// TIA Portal V20 export
FUNCTION "04 T5 EXCENTRIC Transitions" : Void   // FC1418, LAD
TITLE = TRANSITIONS
{ S7_Optimized_Access := 'TRUE' }
// stored: AutoNumber false, SetENOAutomatically false
   VAR_TEMP
      Aux_real : Real;
   END_VAR
BEGIN

REGION Network 1: ============ TRANSITIONS ============
END_REGION

REGION Network 2: Transitions - Zone Status
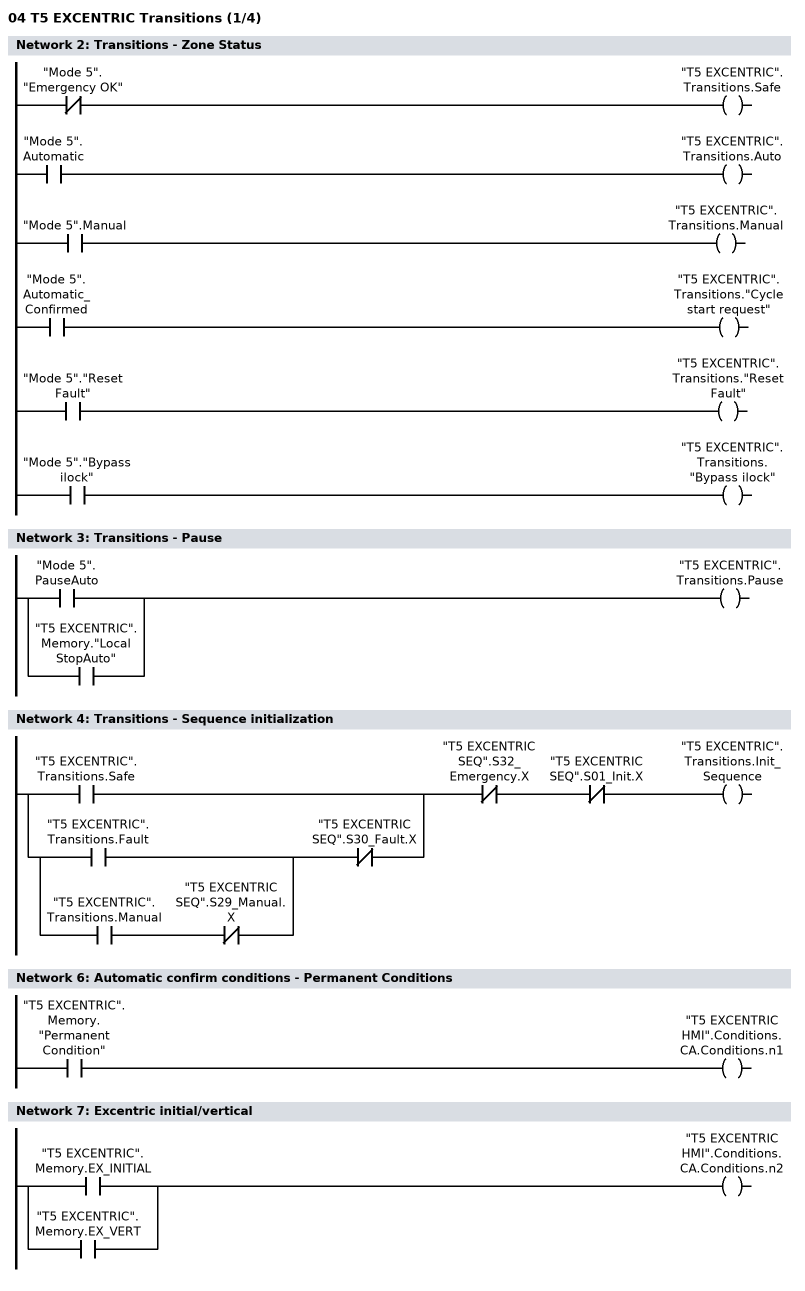
   RUNG wire#powerrail
      I_Contact( "Mode 5"."Emergency OK" )
      Coil( "T5 EXCENTRIC".Transitions.Safe )
   END_RUNG
   RUNG wire#powerrail
      Contact( "Mode 5".Automatic )
      Coil( "T5 EXCENTRIC".Transitions.Auto )
   END_RUNG
   RUNG wire#powerrail
      Contact( "Mode 5".Manual )
      Coil( "T5 EXCENTRIC".Transitions.Manual )
   END_RUNG
   RUNG wire#powerrail
      Contact( "Mode 5".Automatic_Confirmed )
      Coil( "T5 EXCENTRIC".Transitions."Cycle start request" )
   END_RUNG
   RUNG wire#powerrail
      Contact( "Mode 5"."Reset Fault" )
      Coil( "T5 EXCENTRIC".Transitions."Reset Fault" )
   END_RUNG
   RUNG wire#powerrail
      Contact( "Mode 5"."Bypass ilock" )
      Coil( "T5 EXCENTRIC".Transitions."Bypass ilock" )
   END_RUNG
   // the same network as SCL:
   "T5 EXCENTRIC".Transitions.Safe := NOT "Mode 5"."Emergency OK";
   "T5 EXCENTRIC".Transitions.Auto := "Mode 5".Automatic;
   "T5 EXCENTRIC".Transitions.Manual := "Mode 5".Manual;
   "T5 EXCENTRIC".Transitions."Cycle start request" := "Mode 5".Automatic_Confirmed;
   "T5 EXCENTRIC".Transitions."Reset Fault" := "Mode 5"."Reset Fault";
   "T5 EXCENTRIC".Transitions."Bypass ilock" := "Mode 5"."Bypass ilock";
END_REGION

REGION Network 3: Transitions - Pause
   RUNG wire#powerrail
      Contact( "Mode 5".PauseAuto )
      wire#w1
      Coil( "T5 EXCENTRIC".Transitions.Pause )
   END_RUNG
   RUNG wire#powerrail
      Contact( "T5 EXCENTRIC".Memory."Local StopAuto" )
   END_RUNG wire#w1
   // the same network as SCL:
   "T5 EXCENTRIC".Transitions.Pause := "Mode 5".PauseAuto OR "T5 EXCENTRIC".Memory."Local StopAuto";
END_REGION

REGION Network 4: Transitions - Sequence initialization
   RUNG wire#powerrail
      Contact( "T5 EXCENTRIC".Transitions.Safe )
      wire#w1
      I_Contact( "T5 EXCENTRIC SEQ".S32_Emergency.X )
      I_Contact( "T5 EXCENTRIC SEQ".S01_Init.X )
      Coil( "T5 EXCENTRIC".Transitions.Init_Sequence )
   END_RUNG
   RUNG wire#powerrail
      Contact( "T5 EXCENTRIC".Transitions.Fault )
      wire#w2
      I_Contact( "T5 EXCENTRIC SEQ".S30_Fault.X )
   END_RUNG wire#w1
   RUNG wire#powerrail
      Contact( "T5 EXCENTRIC".Transitions.Manual )
      I_Contact( "T5 EXCENTRIC SEQ".S29_Manual.X )
   END_RUNG wire#w2
   // the same network as SCL:
   "T5 EXCENTRIC".Transitions.Init_Sequence := ("T5 EXCENTRIC".Transitions.Safe OR (("T5 EXCENTRIC".Transitions.Fault OR ("T5 EXCENTRIC".Transitions.Manual AND NOT "T5 EXCENTRIC SEQ".S29_Manual.X)) AND NOT "T5 EXCENTRIC SEQ".S30_Fault.X)) AND NOT "T5 EXCENTRIC SEQ".S32_Emergency.X AND NOT "T5 EXCENTRIC SEQ".S01_Init.X;
END_REGION

REGION Network 5: ============ AUTOMATIC CONFIRM CONDITIONS - 1ST PIECE ============
END_REGION

REGION Network 6: Automatic confirm conditions - Permanent Conditions
   RUNG wire#powerrail
      Contact( "T5 EXCENTRIC".Memory."Permanent Condition" )
      Coil( "T5 EXCENTRIC HMI".Conditions.CA.Conditions.n1 )
   END_RUNG
   // the same network as SCL:
   "T5 EXCENTRIC HMI".Conditions.CA.Conditions.n1 := "T5 EXCENTRIC".Memory."Permanent Condition";
END_REGION

REGION Network 7: Excentric initial/vertical
   RUNG wire#powerrail
      Contact( "T5 EXCENTRIC".Memory.EX_INITIAL )
      wire#w1
      Coil( "T5 EXCENTRIC HMI".Conditions.CA.Conditions.n2 )
   END_RUNG
   RUNG wire#powerrail
      Contact( "T5 EXCENTRIC".Memory.EX_VERT )
   END_RUNG wire#w1
   // the same network as SCL:
   "T5 EXCENTRIC HMI".Conditions.CA.Conditions.n2 := "T5 EXCENTRIC".Memory.EX_INITIAL OR "T5 EXCENTRIC".Memory.EX_VERT;
END_REGION

REGION Network 8: Transitions - First Piece
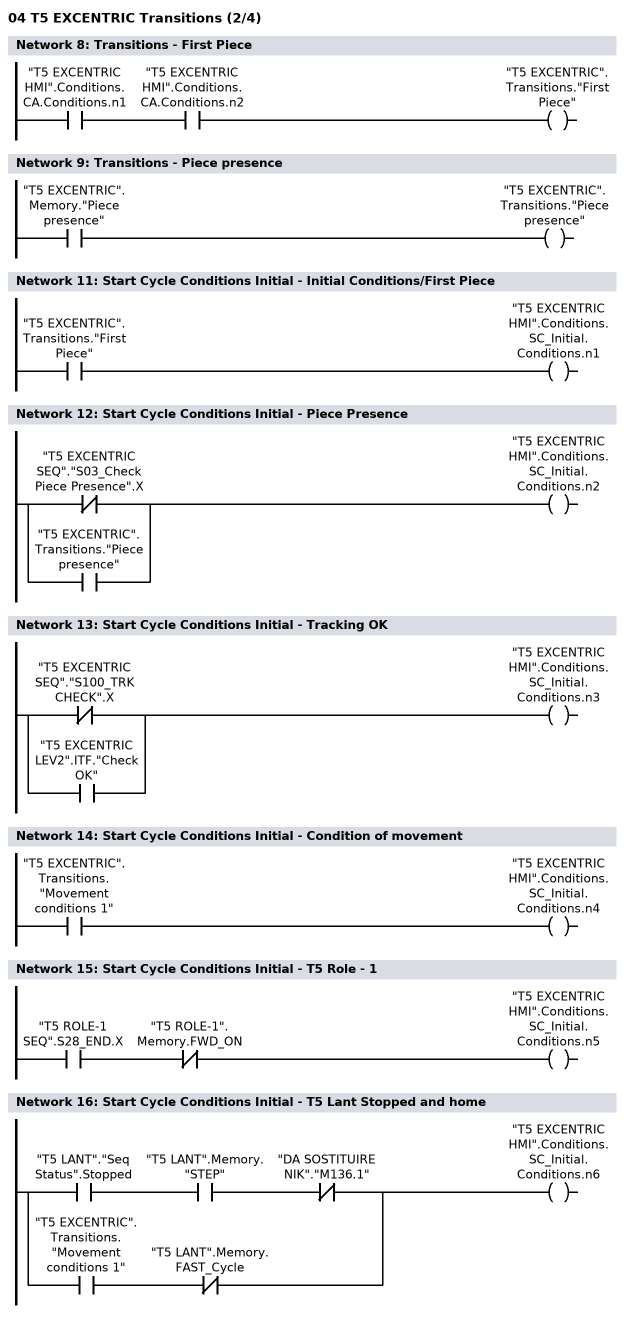
   RUNG wire#powerrail
      Contact( "T5 EXCENTRIC HMI".Conditions.CA.Conditions.n1 )
      Contact( "T5 EXCENTRIC HMI".Conditions.CA.Conditions.n2 )
      Coil( "T5 EXCENTRIC".Transitions."First Piece" )
   END_RUNG
   // the same network as SCL:
   "T5 EXCENTRIC".Transitions."First Piece" := "T5 EXCENTRIC HMI".Conditions.CA.Conditions.n1 AND "T5 EXCENTRIC HMI".Conditions.CA.Conditions.n2;
END_REGION

REGION Network 9: Transitions - Piece presence
   RUNG wire#powerrail
      Contact( "T5 EXCENTRIC".Memory."Piece presence" )
      Coil( "T5 EXCENTRIC".Transitions."Piece presence" )
   END_RUNG
   // the same network as SCL:
   "T5 EXCENTRIC".Transitions."Piece presence" := "T5 EXCENTRIC".Memory."Piece presence";
END_REGION

REGION Network 10: ============ START CYCLE CONDITIONS INITIAL ============
END_REGION

REGION Network 11: Start Cycle Conditions Initial - Initial Conditions/First Piece
   RUNG wire#powerrail
      Contact( "T5 EXCENTRIC".Transitions."First Piece" )
      Coil( "T5 EXCENTRIC HMI".Conditions.SC_Initial.Conditions.n1 )
   END_RUNG
   // the same network as SCL:
   "T5 EXCENTRIC HMI".Conditions.SC_Initial.Conditions.n1 := "T5 EXCENTRIC".Transitions."First Piece";
END_REGION

REGION Network 12: Start Cycle Conditions Initial - Piece Presence
   RUNG wire#powerrail
      I_Contact( "T5 EXCENTRIC SEQ"."S03_Check Piece Presence".X )
      wire#w1
      Coil( "T5 EXCENTRIC HMI".Conditions.SC_Initial.Conditions.n2 )
   END_RUNG
   RUNG wire#powerrail
      Contact( "T5 EXCENTRIC".Transitions."Piece presence" )
   END_RUNG wire#w1
   // the same network as SCL:
   "T5 EXCENTRIC HMI".Conditions.SC_Initial.Conditions.n2 := NOT "T5 EXCENTRIC SEQ"."S03_Check Piece Presence".X OR "T5 EXCENTRIC".Transitions."Piece presence";
END_REGION

REGION Network 13: Start Cycle Conditions Initial - Tracking OK
   RUNG wire#powerrail
      I_Contact( "T5 EXCENTRIC SEQ"."S100_TRK CHECK".X )
      wire#w1
      Coil( "T5 EXCENTRIC HMI".Conditions.SC_Initial.Conditions.n3 )
   END_RUNG
   RUNG wire#powerrail
      Contact( "T5 EXCENTRIC LEV2".ITF."Check OK" )
   END_RUNG wire#w1
   // the same network as SCL:
   "T5 EXCENTRIC HMI".Conditions.SC_Initial.Conditions.n3 := NOT "T5 EXCENTRIC SEQ"."S100_TRK CHECK".X OR "T5 EXCENTRIC LEV2".ITF."Check OK";
END_REGION

REGION Network 14: Start Cycle Conditions Initial - Condition of movement
   RUNG wire#powerrail
      Contact( "T5 EXCENTRIC".Transitions."Movement conditions 1" )
      Coil( "T5 EXCENTRIC HMI".Conditions.SC_Initial.Conditions.n4 )
   END_RUNG
   // the same network as SCL:
   "T5 EXCENTRIC HMI".Conditions.SC_Initial.Conditions.n4 := "T5 EXCENTRIC".Transitions."Movement conditions 1";
END_REGION

REGION Network 15: Start Cycle Conditions Initial - T5 Role - 1
   RUNG wire#powerrail
      Contact( "T5 ROLE-1 SEQ".S28_END.X )
      I_Contact( "T5 ROLE-1".Memory.FWD_ON )
      Coil( "T5 EXCENTRIC HMI".Conditions.SC_Initial.Conditions.n5 )
   END_RUNG
   // the same network as SCL:
   "T5 EXCENTRIC HMI".Conditions.SC_Initial.Conditions.n5 := "T5 ROLE-1 SEQ".S28_END.X AND NOT "T5 ROLE-1".Memory.FWD_ON;
END_REGION

REGION Network 16: Start Cycle Conditions Initial - T5 Lant Stopped and home
   RUNG wire#powerrail
      Contact( "T5 LANT"."Seq Status".Stopped )
      Contact( "T5 LANT".Memory."STEP" )
      I_Contact( "DA SOSTITUIRE NIK"."M136.1" )
      wire#w1
      Coil( "T5 EXCENTRIC HMI".Conditions.SC_Initial.Conditions.n6 )
   END_RUNG
   RUNG wire#powerrail
      Contact( "T5 EXCENTRIC".Transitions."Movement conditions 1" )
      I_Contact( "T5 LANT".Memory.FAST_Cycle )
   END_RUNG wire#w1
   // the same network as SCL:
   "T5 EXCENTRIC HMI".Conditions.SC_Initial.Conditions.n6 := ("T5 LANT"."Seq Status".Stopped AND "T5 LANT".Memory."STEP" AND NOT "DA SOSTITUIRE NIK"."M136.1") OR ("T5 EXCENTRIC".Transitions."Movement conditions 1" AND NOT "T5 LANT".Memory.FAST_Cycle);
END_REGION

REGION Network 17: Start Cycle Conditions Initial - T5 Lant free
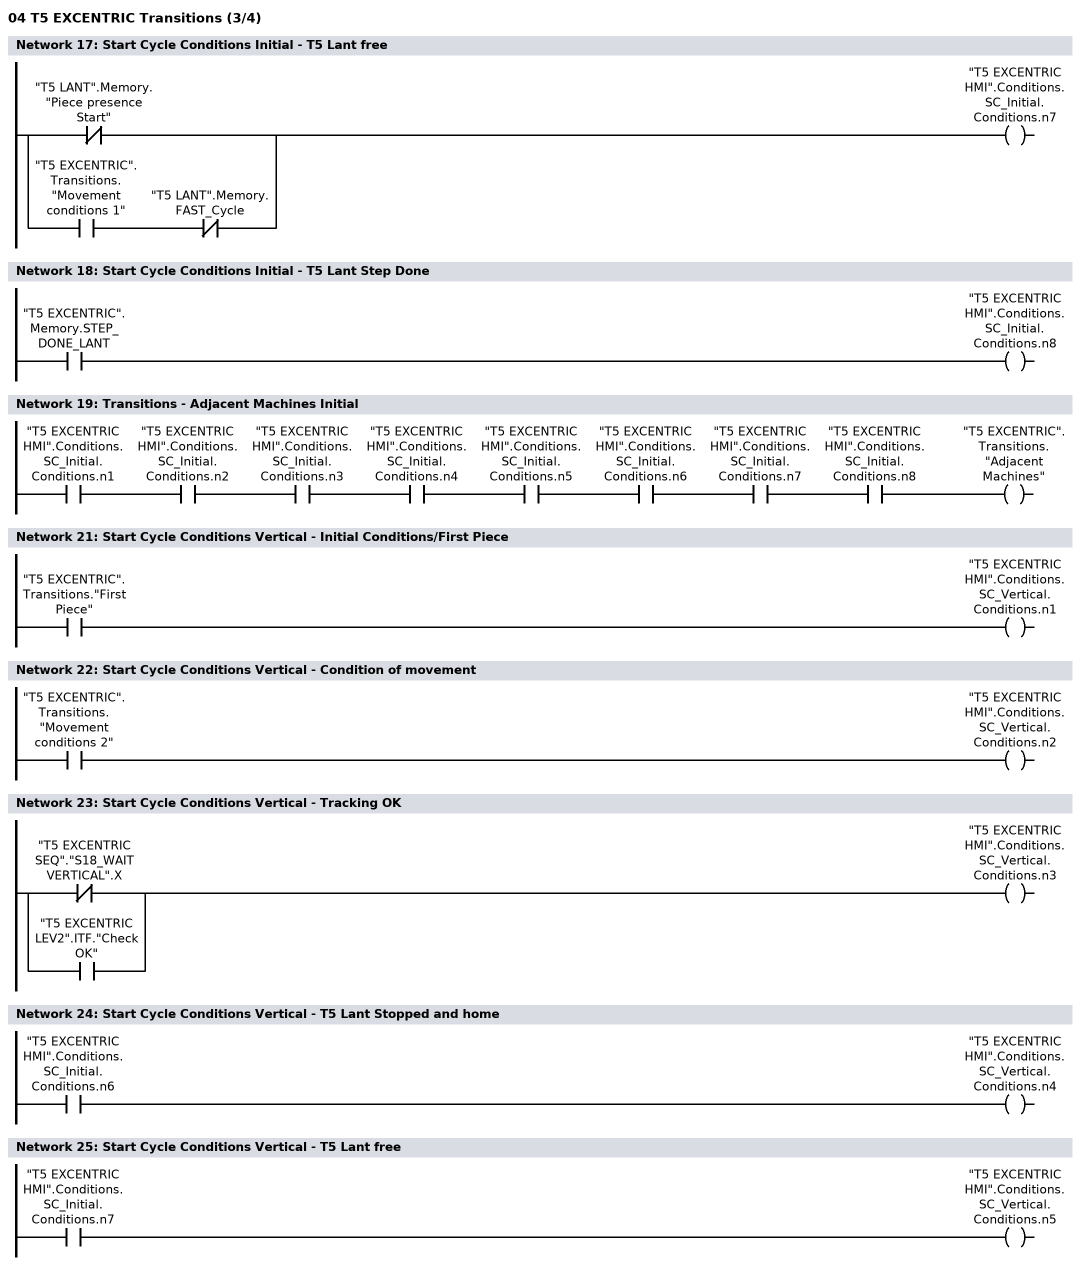
   RUNG wire#powerrail
      I_Contact( "T5 LANT".Memory."Piece presence Start" )
      wire#w1
      Coil( "T5 EXCENTRIC HMI".Conditions.SC_Initial.Conditions.n7 )
   END_RUNG
   RUNG wire#powerrail
      Contact( "T5 EXCENTRIC".Transitions."Movement conditions 1" )
      I_Contact( "T5 LANT".Memory.FAST_Cycle )
   END_RUNG wire#w1
   // the same network as SCL:
   "T5 EXCENTRIC HMI".Conditions.SC_Initial.Conditions.n7 := NOT "T5 LANT".Memory."Piece presence Start" OR ("T5 EXCENTRIC".Transitions."Movement conditions 1" AND NOT "T5 LANT".Memory.FAST_Cycle);
END_REGION

REGION Network 18: Start Cycle Conditions Initial - T5 Lant Step Done
   RUNG wire#powerrail
      Contact( "T5 EXCENTRIC".Memory.STEP_DONE_LANT )
      Coil( "T5 EXCENTRIC HMI".Conditions.SC_Initial.Conditions.n8 )
   END_RUNG
   // the same network as SCL:
   "T5 EXCENTRIC HMI".Conditions.SC_Initial.Conditions.n8 := "T5 EXCENTRIC".Memory.STEP_DONE_LANT;
END_REGION

REGION Network 19: Transitions - Adjacent Machines Initial
   RUNG wire#powerrail
      Contact( "T5 EXCENTRIC HMI".Conditions.SC_Initial.Conditions.n1 )
      Contact( "T5 EXCENTRIC HMI".Conditions.SC_Initial.Conditions.n2 )
      Contact( "T5 EXCENTRIC HMI".Conditions.SC_Initial.Conditions.n3 )
      Contact( "T5 EXCENTRIC HMI".Conditions.SC_Initial.Conditions.n4 )
      Contact( "T5 EXCENTRIC HMI".Conditions.SC_Initial.Conditions.n5 )
      Contact( "T5 EXCENTRIC HMI".Conditions.SC_Initial.Conditions.n6 )
      Contact( "T5 EXCENTRIC HMI".Conditions.SC_Initial.Conditions.n7 )
      Contact( "T5 EXCENTRIC HMI".Conditions.SC_Initial.Conditions.n8 )
      Coil( "T5 EXCENTRIC".Transitions."Adjacent Machines" )
   END_RUNG
   // the same network as SCL:
   "T5 EXCENTRIC".Transitions."Adjacent Machines" := "T5 EXCENTRIC HMI".Conditions.SC_Initial.Conditions.n1 AND "T5 EXCENTRIC HMI".Conditions.SC_Initial.Conditions.n2 AND "T5 EXCENTRIC HMI".Conditions.SC_Initial.Conditions.n3 AND "T5 EXCENTRIC HMI".Conditions.SC_Initial.Conditions.n4 AND "T5 EXCENTRIC HMI".Conditions.SC_Initial.Conditions.n5 AND "T5 EXCENTRIC HMI".Conditions.SC_Initial.Conditions.n6 AND "T5 EXCENTRIC HMI".Conditions.SC_Initial.Conditions.n7 AND "T5 EXCENTRIC HMI".Conditions.SC_Initial.Conditions.n8;
END_REGION

REGION Network 20: ============ START CYCLE CONDITIONS VERTICAL ============
END_REGION

REGION Network 21: Start Cycle Conditions Vertical - Initial Conditions/First Piece
   RUNG wire#powerrail
      Contact( "T5 EXCENTRIC".Transitions."First Piece" )
      Coil( "T5 EXCENTRIC HMI".Conditions.SC_Vertical.Conditions.n1 )
   END_RUNG
   // the same network as SCL:
   "T5 EXCENTRIC HMI".Conditions.SC_Vertical.Conditions.n1 := "T5 EXCENTRIC".Transitions."First Piece";
END_REGION

REGION Network 22: Start Cycle Conditions Vertical - Condition of movement
   RUNG wire#powerrail
      Contact( "T5 EXCENTRIC".Transitions."Movement conditions 2" )
      Coil( "T5 EXCENTRIC HMI".Conditions.SC_Vertical.Conditions.n2 )
   END_RUNG
   // the same network as SCL:
   "T5 EXCENTRIC HMI".Conditions.SC_Vertical.Conditions.n2 := "T5 EXCENTRIC".Transitions."Movement conditions 2";
END_REGION

REGION Network 23: Start Cycle Conditions Vertical - Tracking OK
   RUNG wire#powerrail
      I_Contact( "T5 EXCENTRIC SEQ"."S18_WAIT VERTICAL".X )
      wire#w1
      Coil( "T5 EXCENTRIC HMI".Conditions.SC_Vertical.Conditions.n3 )
   END_RUNG
   RUNG wire#powerrail
      Contact( "T5 EXCENTRIC LEV2".ITF."Check OK" )
   END_RUNG wire#w1
   // the same network as SCL:
   "T5 EXCENTRIC HMI".Conditions.SC_Vertical.Conditions.n3 := NOT "T5 EXCENTRIC SEQ"."S18_WAIT VERTICAL".X OR "T5 EXCENTRIC LEV2".ITF."Check OK";
END_REGION

REGION Network 24: Start Cycle Conditions Vertical - T5 Lant Stopped and home
   RUNG wire#powerrail
      Contact( "T5 EXCENTRIC HMI".Conditions.SC_Initial.Conditions.n6 )
      Coil( "T5 EXCENTRIC HMI".Conditions.SC_Vertical.Conditions.n4 )
   END_RUNG
   // the same network as SCL:
   "T5 EXCENTRIC HMI".Conditions.SC_Vertical.Conditions.n4 := "T5 EXCENTRIC HMI".Conditions.SC_Initial.Conditions.n6;
END_REGION

REGION Network 25: Start Cycle Conditions Vertical - T5 Lant free
   RUNG wire#powerrail
      Contact( "T5 EXCENTRIC HMI".Conditions.SC_Initial.Conditions.n7 )
      Coil( "T5 EXCENTRIC HMI".Conditions.SC_Vertical.Conditions.n5 )
   END_RUNG
   // the same network as SCL:
   "T5 EXCENTRIC HMI".Conditions.SC_Vertical.Conditions.n5 := "T5 EXCENTRIC HMI".Conditions.SC_Initial.Conditions.n7;
END_REGION

REGION Network 26: Start Cycle Conditions Vertical - T5 Lant Step Done
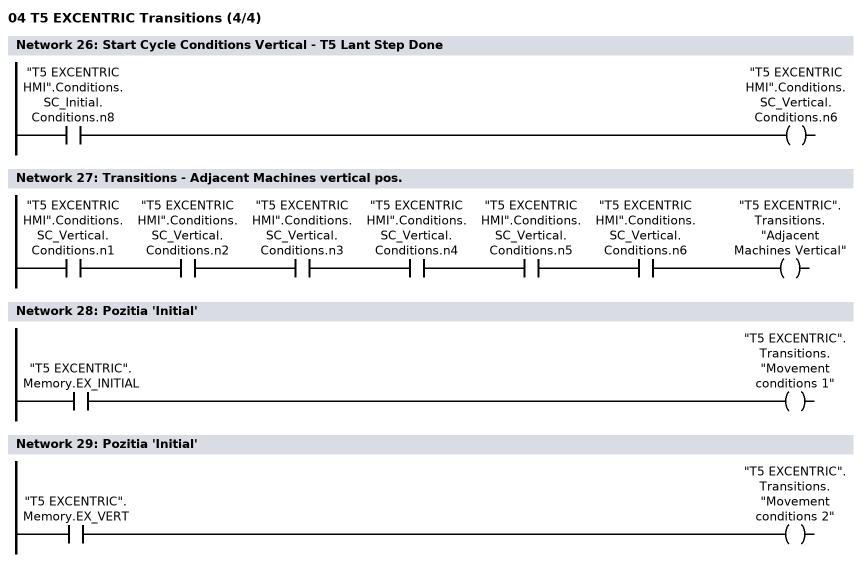
   RUNG wire#powerrail
      Contact( "T5 EXCENTRIC HMI".Conditions.SC_Initial.Conditions.n8 )
      Coil( "T5 EXCENTRIC HMI".Conditions.SC_Vertical.Conditions.n6 )
   END_RUNG
   // the same network as SCL:
   "T5 EXCENTRIC HMI".Conditions.SC_Vertical.Conditions.n6 := "T5 EXCENTRIC HMI".Conditions.SC_Initial.Conditions.n8;
END_REGION

REGION Network 27: Transitions - Adjacent Machines vertical pos.
   RUNG wire#powerrail
      Contact( "T5 EXCENTRIC HMI".Conditions.SC_Vertical.Conditions.n1 )
      Contact( "T5 EXCENTRIC HMI".Conditions.SC_Vertical.Conditions.n2 )
      Contact( "T5 EXCENTRIC HMI".Conditions.SC_Vertical.Conditions.n3 )
      Contact( "T5 EXCENTRIC HMI".Conditions.SC_Vertical.Conditions.n4 )
      Contact( "T5 EXCENTRIC HMI".Conditions.SC_Vertical.Conditions.n5 )
      Contact( "T5 EXCENTRIC HMI".Conditions.SC_Vertical.Conditions.n6 )
      Coil( "T5 EXCENTRIC".Transitions."Adjacent Machines Vertical" )
   END_RUNG
   // the same network as SCL:
   "T5 EXCENTRIC".Transitions."Adjacent Machines Vertical" := "T5 EXCENTRIC HMI".Conditions.SC_Vertical.Conditions.n1 AND "T5 EXCENTRIC HMI".Conditions.SC_Vertical.Conditions.n2 AND "T5 EXCENTRIC HMI".Conditions.SC_Vertical.Conditions.n3 AND "T5 EXCENTRIC HMI".Conditions.SC_Vertical.Conditions.n4 AND "T5 EXCENTRIC HMI".Conditions.SC_Vertical.Conditions.n5 AND "T5 EXCENTRIC HMI".Conditions.SC_Vertical.Conditions.n6;
END_REGION

REGION Network 28: Pozitia 'Initial'
   RUNG wire#powerrail
      Contact( "T5 EXCENTRIC".Memory.EX_INITIAL )
      Coil( "T5 EXCENTRIC".Transitions."Movement conditions 1" )
   END_RUNG
   // the same network as SCL:
   "T5 EXCENTRIC".Transitions."Movement conditions 1" := "T5 EXCENTRIC".Memory.EX_INITIAL;
END_REGION

REGION Network 29: Pozitia 'Initial'
   RUNG wire#powerrail
      Contact( "T5 EXCENTRIC".Memory.EX_VERT )
      Coil( "T5 EXCENTRIC".Transitions."Movement conditions 2" )
   END_RUNG
   // the same network as SCL:
   "T5 EXCENTRIC".Transitions."Movement conditions 2" := "T5 EXCENTRIC".Memory.EX_VERT;
END_REGION
END_FUNCTION
